(* IEC 61131-3 sources: TIA2AX/tests/V19/test_projects/expected/HW_2200330/ST20_PLC, 7 files *)

(* ---- HwIdentifiers.st ---- *)
TYPE
	HwIdentifiers : WORD
	(
		ST20_PLC_Profilschiene_0 :=	WORD#256,
		ST20_PLC :=	WORD#48,
		ST20_PLC_Card_reader_writer_1 :=	WORD#51,
		ST20_PLC_CPU_display_1 :=	WORD#54,
		ST20_PLC_OPC_UA_1 :=	WORD#117,
		ST20_PLC_DP_interface_1 :=	WORD#60,
		ST20_PLC_PROFINET_interface_1 :=	WORD#64,
		ST20_PLC_PROFINET_interface_1_Port_1 :=	WORD#65,
		ST20_PLC_PROFINET_interface_1_Port_2 :=	WORD#66,
		ST20_PLC_PROFINET_interface_2 :=	WORD#72,
		ST20_PLC_PROFINET_interface_2_Port_1 :=	WORD#73,
		ST20_Switch_SCALANCE_X_rack :=	WORD#544,
		ST20_Switch :=	WORD#545,
		ST20_Switch_ST20_Switch :=	WORD#546,
		ST20_Switch_SCALANCE_interface_1 :=	WORD#547,
		ST20_Switch_SCALANCE_interface_1_Port_1 :=	WORD#548,
		ST20_Switch_SCALANCE_interface_1_Port_2 :=	WORD#549,
		ST20_Switch_SCALANCE_interface_1_Port_3 :=	WORD#550,
		ST20_Switch_SCALANCE_interface_1_Port_4 :=	WORD#551,
		ST20_Switch_SCALANCE_interface_1_Port_5 :=	WORD#552,
		ST20_Switch_SCALANCE_interface_1_Port_6 :=	WORD#553,
		ST20_Switch_SCALANCE_interface_1_Port_7 :=	WORD#554,
		ST20_Switch_SCALANCE_interface_1_Port_8 :=	WORD#555,
		ST20_Switch_SCALANCE_interface_1_Port_9 :=	WORD#556,
		ST20_Switch_SCALANCE_interface_1_Port_10 :=	WORD#557,
		ST20_Switch_SCALANCE_interface_1_Port_11 :=	WORD#558,
		ST20_Switch_SCALANCE_interface_1_Port_12 :=	WORD#559,
		ST20_Switch_SCALANCE_interface_1_Port_13 :=	WORD#560,
		ST20_Switch_SCALANCE_interface_1_Port_14 :=	WORD#561,
		ST20_Switch_SCALANCE_interface_1_Port_15 :=	WORD#562,
		ST20_Switch_SCALANCE_interface_1_Port_16 :=	WORD#563,
		ST20_Switch_2_SCALANCE_X_rack :=	WORD#565,
		ST20_Switch_2 :=	WORD#566,
		ST20_Switch_2_ST20_Switch_2 :=	WORD#567,
		ST20_Switch_2_SCALANCE_interface_1 :=	WORD#568,
		ST20_Switch_2_SCALANCE_interface_1_Port_1 :=	WORD#569,
		ST20_Switch_2_SCALANCE_interface_1_Port_2 :=	WORD#570,
		ST20_Switch_2_SCALANCE_interface_1_Port_3 :=	WORD#571,
		ST20_Switch_2_SCALANCE_interface_1_Port_4 :=	WORD#572,
		ST20_Switch_2_SCALANCE_interface_1_Port_5 :=	WORD#573,
		ST20_Switch_2_SCALANCE_interface_1_Port_6 :=	WORD#574,
		ST20_Switch_2_SCALANCE_interface_1_Port_7 :=	WORD#575,
		ST20_Switch_2_SCALANCE_interface_1_Port_8 :=	WORD#576,
		ST20_Switch_2_SCALANCE_interface_1_Port_9 :=	WORD#577,
		ST20_Switch_2_SCALANCE_interface_1_Port_10 :=	WORD#578,
		ST20_Switch_2_SCALANCE_interface_1_Port_11 :=	WORD#579,
		ST20_Switch_2_SCALANCE_interface_1_Port_12 :=	WORD#580,
		ST20_Switch_2_SCALANCE_interface_1_Port_13 :=	WORD#581,
		ST20_Switch_2_SCALANCE_interface_1_Port_14 :=	WORD#582,
		ST20_Switch_2_SCALANCE_interface_1_Port_15 :=	WORD#583,
		ST20_Switch_2_SCALANCE_interface_1_Port_16 :=	WORD#584,
		ST20_Switch_3_SCALANCE_X_rack :=	WORD#586,
		ST20_Switch_3 :=	WORD#587,
		ST20_Switch_3_ST20_Switch_3 :=	WORD#588,
		ST20_Switch_3_SCALANCE_interface_1 :=	WORD#589,
		ST20_Switch_3_SCALANCE_interface_1_Port_1 :=	WORD#590,
		ST20_Switch_3_SCALANCE_interface_1_Port_2 :=	WORD#591,
		ST20_Switch_3_SCALANCE_interface_1_Port_3 :=	WORD#592,
		ST20_Switch_3_SCALANCE_interface_1_Port_4 :=	WORD#593,
		ST20_Switch_3_SCALANCE_interface_1_Port_5 :=	WORD#594,
		ST20_Switch_3_SCALANCE_interface_1_Port_6 :=	WORD#595,
		ST20_Switch_3_SCALANCE_interface_1_Port_7 :=	WORD#596,
		ST20_Switch_3_SCALANCE_interface_1_Port_8 :=	WORD#597,
		ST20_HMI_ConnectionBox_Connection_Box :=	WORD#265,
		ST20_HMI_ConnectionBox :=	WORD#258,
		ST20_HMI_ConnectionBox_ST20_HMI_ConnectionBox :=	WORD#259,
		ST20_HMI_ConnectionBox_SCALANCE_interface_1 :=	WORD#260,
		ST20_HMI_ConnectionBox_SCALANCE_interface_1_Port_1 :=	WORD#261,
		ST20_HMI_ConnectionBox_SCALANCE_interface_1_Port_2 :=	WORD#262,
		ST20_HMI_ConnectionBox_SCALANCE_interface_1_Port_3 :=	WORD#263,
		ST20_CPX_PN_IO_Interface :=	WORD#271,
		ST20_CPX_PN_IO_Interface_Port_1 :=	WORD#272,
		ST20_CPX_PN_IO_Interface_Port_2 :=	WORD#273,
		ST20_CPX_CPX :=	WORD#274,
		ST20_CPX_MPA1S_VMPA1_FB_EMS_8_8DO_1 :=	WORD#275,
		ST20_CPX_MPA1S_VMPA1_FB_EMS_8_8DO_2 :=	WORD#276,
		ST20_CPX_MPA1S_VMPA1_FB_EMS_8_8DO_3 :=	WORD#277,
		ST20_CPX_MPA1S_VMPA1_FB_EMS_8_8DO_4 :=	WORD#266,
		ST20_CPX_MPA1G_VMPA1_FB_EMG_8_8DO_1 :=	WORD#267,
		ST20_6_Promess_Rack :=	WORD#328,
		ST20_6_Promess :=	WORD#329,
		ST20_6_Promess_X1 :=	WORD#330,
		ST20_6_Promess_X1_X1_P1 :=	WORD#331,
		ST20_6_Promess_X1_X1_P2 :=	WORD#332,
		ST20_6_Promess_UniDrive_M :=	WORD#333,
		ST20_6_Promess_Menu_30_01_In_1 :=	WORD#334,
		ST20_6_Promess_Menu_30_02_In_1 :=	WORD#335,
		ST20_6_Promess_Menu_30_03_In_1 :=	WORD#336,
		ST20_6_Promess_Menu_30_04_In_1 :=	WORD#337,
		ST20_6_Promess_Menu_30_05_In_1 :=	WORD#338,
		ST20_6_Promess_Menu_30_06_In_1 :=	WORD#339,
		ST20_6_Promess_Menu_30_07_In_1 :=	WORD#340,
		ST20_6_Promess_Menu_30_08_In_1 :=	WORD#341,
		ST20_6_Promess_Menu_30_09_In_1 :=	WORD#342,
		ST20_6_Promess_Menu_30_10_In_1 :=	WORD#343,
		ST20_6_Promess_Menu_30_11_In_1 :=	WORD#344,
		ST20_6_Promess_Menu_30_12_In_1 :=	WORD#345,
		ST20_6_Promess_Menu_30_13_In_1 :=	WORD#346,
		ST20_6_Promess_Menu_30_14_In_1 :=	WORD#347,
		ST20_6_Promess_Menu_30_15_In_1 :=	WORD#348,
		ST20_6_Promess_Menu_30_16_In_1 :=	WORD#278,
		ST20_6_Promess_Menu_30_33_Out_1 :=	WORD#279,
		ST20_6_Promess_Menu_30_34_Out_1 :=	WORD#280,
		ST20_6_Promess_Menu_30_35_Out_1 :=	WORD#281,
		ST20_6_Promess_Menu_30_36_Out_1 :=	WORD#282,
		ST20_6_Promess_Menu_30_37_Out_1 :=	WORD#283,
		ST20_6_Promess_Menu_30_38_Out_1 :=	WORD#284,
		ST20_6_Promess_Menu_30_39_Out_1 :=	WORD#285,
		ST20_6_Promess_Menu_30_40_Out_1 :=	WORD#286,
		ST20_6_Promess_Menu_30_41_Out_1 :=	WORD#287,
		ST20_6_Promess_Menu_30_42_Out_1 :=	WORD#288,
		ST20_6_Promess_Menu_30_43_Out_1 :=	WORD#289,
		ST20_6_Promess_Menu_30_44_Out_1 :=	WORD#290,
		ST20_6_Promess_Menu_30_45_Out_1 :=	WORD#291,
		ST20_6_Promess_Menu_30_46_Out_1 :=	WORD#292,
		ST20_6_Promess_Menu_30_47_Out_1 :=	WORD#293,
		ST20_6_Promess_Menu_30_48_Out_1 :=	WORD#294,
		ST20_6_Promess_Menu_30_17_In_1 :=	WORD#295,
		ST20_6_Promess_Menu_30_18_In_1 :=	WORD#296,
		ST20_6_Promess_Menu_30_19_In_1 :=	WORD#297,
		ST20_6_Promess_Menu_30_20_In_1 :=	WORD#298,
		ST20_6_Promess_Menu_30_21_In_1 :=	WORD#299,
		ST20_6_Promess_Menu_30_22_In_1 :=	WORD#300,
		ST20_6_Promess_Menu_30_23_In_1 :=	WORD#301,
		ST20_6_Promess_Menu_30_24_In_1 :=	WORD#302,
		ST20_6_Promess_Menu_30_25_In_1 :=	WORD#303,
		ST20_6_Promess_Menu_30_26_In_1 :=	WORD#304,
		ST20_6_Promess_Menu_30_27_In_1 :=	WORD#305,
		ST20_6_Promess_Menu_30_28_In_1 :=	WORD#306,
		ST20_6_Promess_Menu_30_29_In_1 :=	WORD#307,
		ST20_6_Promess_Menu_30_30_In_1 :=	WORD#308,
		ST20_6_Promess_Menu_30_31_In_1 :=	WORD#309,
		ST20_6_Promess_Menu_30_32_In_1 :=	WORD#310,
		ST20_6_Promess_Menu_30_49_Out_1 :=	WORD#311,
		ST20_6_Promess_Menu_30_50_Out_1 :=	WORD#312,
		ST20_6_Promess_Menu_30_51_Out_1 :=	WORD#313,
		ST20_6_Promess_Menu_30_52_Out_1 :=	WORD#314,
		ST20_6_Promess_Menu_30_53_Out_1 :=	WORD#315,
		ST20_6_Promess_Menu_30_54_Out_1 :=	WORD#316,
		ST20_6_Promess_Menu_30_55_Out_1 :=	WORD#317,
		ST20_6_Promess_Menu_30_56_Out_1 :=	WORD#318,
		ST20_6_Promess_Menu_30_57_Out_1 :=	WORD#319,
		ST20_6_Promess_Menu_30_58_Out_1 :=	WORD#320,
		ST20_6_Promess_Menu_30_59_Out_1 :=	WORD#321,
		ST20_6_Promess_Menu_30_60_Out_1 :=	WORD#322,
		ST20_6_Promess_Menu_30_61_Out_1 :=	WORD#323,
		ST20_6_Promess_Menu_30_62_Out_1 :=	WORD#324,
		ST20_6_Promess_Menu_30_63_Out_1 :=	WORD#325,
		ST20_6_Promess_Menu_30_64_Out_1 :=	WORD#326,
		ST20_7_CMMT_3GF1_PN_IO_Interface :=	WORD#352,
		ST20_7_CMMT_3GF1_PN_IO_Interface_Port_1 :=	WORD#353,
		ST20_7_CMMT_3GF1_PN_IO_Interface_Port_2 :=	WORD#354,
		ST20_7_CMMT_3GF1_CMMT_AS_V1 :=	WORD#355,
		ST20_7_CMMT_3GF1_DO_SERVO_1_Module_Access_Point :=	WORD#357,
		ST20_7_CMMT_3GF1_DO_SERVO_1_Siemens_telegram_111_PZD_12_12 :=	WORD#358,
		ST20_7_CMMT_3GF1_Siemens_telegram_111_PZD_12_12 :=	WORD#358,
		ST20_1_DM260_Rack :=	WORD#360,
		ST20_1_DM260 :=	WORD#361,
		ST20_1_DM260_Interface :=	WORD#362,
		ST20_1_DM260_Interface_Port_1 :=	WORD#363,
		ST20_1_DM260_DataMan_260 :=	WORD#364,
		ST20_1_DM260_Acquisition_Control_1 :=	WORD#365,
		ST20_1_DM260_Acquisition_Status_1 :=	WORD#366,
		ST20_1_DM260_Results_Control_1 :=	WORD#367,
		ST20_1_DM260_Results_Status_1 :=	WORD#368,
		ST20_1_DM260_Soft_Event_Control_1 :=	WORD#369,
		ST20_1_DM260_User_Data_64_bytes_1 :=	WORD#370,
		ST20_1_DM260_Result_Data_64_bytes_1 :=	WORD#371,
		ST20_5_DM260_Rack :=	WORD#373,
		ST20_5_DM260 :=	WORD#374,
		ST20_5_DM260_Interface :=	WORD#375,
		ST20_5_DM260_Interface_Port_1 :=	WORD#376,
		ST20_5_DM260_DataMan_260 :=	WORD#377,
		ST20_5_DM260_Acquisition_Control_1 :=	WORD#378,
		ST20_5_DM260_Acquisition_Status_1 :=	WORD#379,
		ST20_5_DM260_Results_Control_1 :=	WORD#380,
		ST20_5_DM260_Results_Status_1 :=	WORD#381,
		ST20_5_DM260_Soft_Event_Control_1 :=	WORD#382,
		ST20_5_DM260_User_Data_64_bytes_1 :=	WORD#383,
		ST20_5_DM260_Result_Data_64_bytes_1 :=	WORD#384,
		ST20_2_DM260_Rack :=	WORD#386,
		ST20_2_DM260 :=	WORD#387,
		ST20_2_DM260_Interface :=	WORD#388,
		ST20_2_DM260_Interface_Port_1 :=	WORD#389,
		ST20_2_DM260_DataMan_260 :=	WORD#390,
		ST20_2_DM260_Acquisition_Control_1 :=	WORD#391,
		ST20_2_DM260_Acquisition_Status_1 :=	WORD#392,
		ST20_2_DM260_Results_Control_1 :=	WORD#393,
		ST20_2_DM260_Results_Status_1 :=	WORD#394,
		ST20_2_DM260_Soft_Event_Control_1 :=	WORD#395,
		ST20_2_DM260_User_Data_64_bytes_1 :=	WORD#396,
		ST20_2_DM260_Result_Data_64_bytes_1 :=	WORD#397,
		ST20_2_TZ535_PN_Rack :=	WORD#399,
		ST20_2_TZ535_PN :=	WORD#400,
		ST20_2_TZ535_PN_Interface :=	WORD#401,
		ST20_2_TZ535_PN_Interface_Port_1 :=	WORD#402,
		ST20_2_TZ535_PN_Interface_Port_2 :=	WORD#403,
		ST20_2_TZ535_PN_2D_TZ535_PN_PROFINET_IO :=	WORD#404,
		ST20_2_TZ535_PN_In_Out_32_byte_1 :=	WORD#405,
		ST20_3_TZ535_PN_Rack :=	WORD#407,
		ST20_3_TZ535_PN :=	WORD#408,
		ST20_3_TZ535_PN_Interface :=	WORD#409,
		ST20_3_TZ535_PN_Interface_Port_1 :=	WORD#410,
		ST20_3_TZ535_PN_Interface_Port_2 :=	WORD#411,
		ST20_3_TZ535_PN_2D_TZ535_PN_PROFINET_IO :=	WORD#412,
		ST20_3_TZ535_PN_In_Out_32_byte_1 :=	WORD#413,
		ST20_4_TZ535_PN_Rack :=	WORD#415,
		ST20_4_TZ535_PN :=	WORD#416,
		ST20_4_TZ535_PN_Interface :=	WORD#417,
		ST20_4_TZ535_PN_Interface_Port_1 :=	WORD#418,
		ST20_4_TZ535_PN_Interface_Port_2 :=	WORD#419,
		ST20_4_TZ535_PN_2D_TZ535_PN_PROFINET_IO :=	WORD#420,
		ST20_4_TZ535_PN_In_Out_32_byte_1 :=	WORD#421,
		ST20_5_TZ535_PN_Rack :=	WORD#423,
		ST20_5_TZ535_PN :=	WORD#424,
		ST20_5_TZ535_PN_Interface :=	WORD#425,
		ST20_5_TZ535_PN_Interface_Port_1 :=	WORD#426,
		ST20_5_TZ535_PN_Interface_Port_2 :=	WORD#427,
		ST20_5_TZ535_PN_2D_TZ535_PN_PROFINET_IO :=	WORD#428,
		ST20_5_TZ535_PN_In_Out_32_byte_1 :=	WORD#429,
		ST20_ET200SP_Rack_0 :=	WORD#431,
		ST20_ET200SP :=	WORD#432,
		ST20_ET200SP_ST20_ET200SP :=	WORD#433,
		ST20_ET200SP_PROFINET_interface :=	WORD#434,
		ST20_ET200SP_PROFINET_interface_Port_1 :=	WORD#436,
		ST20_ET200SP_PROFINET_interface_Port_2 :=	WORD#435,
		ST20_ET200SP_BA_2xRJ45 :=	WORD#436,
		ST20_ET200SP_CM_4xIO_Link_1 :=	WORD#437,
		ST20_ET200SP_CM_4xIO_Link_2 :=	WORD#438,
		ST20_ET200SP_DI_16x24VDC_ST_1 :=	WORD#439,
		ST20_ET200SP_DI_16x24VDC_ST_2 :=	WORD#440,
		ST20_ET200SP_DI_16x24VDC_ST_3 :=	WORD#441,
		ST20_ET200SP_DI_16x24VDC_ST_4 :=	WORD#442,
		ST20_ET200SP_DQ_16x24VDC_0_5A_ST_1 :=	WORD#443,
		ST20_ET200SP_DQ_16x24VDC_0_5A_ST_2 :=	WORD#444,
		ST20_ET200SP_DQ_16x24VDC_0_5A_ST_3 :=	WORD#445,
		ST20_ET200SP_Servermodul_1 :=	WORD#446,
		ST20_2_Schunk_Rack :=	WORD#448,
		ST20_2_Schunk :=	WORD#449,
		ST20_2_Schunk_Interface :=	WORD#450,
		ST20_2_Schunk_Interface_Port_1 :=	WORD#451,
		ST20_2_Schunk_Interface_Port_2 :=	WORD#452,
		ST20_2_Schunk_DEVICE_SFP :=	WORD#453,
		ST20_2_Schunk_IN_4_Double_Words_1 :=	WORD#454,
		ST20_2_Schunk_OUT_4_Double_Words_1 :=	WORD#455,
		ST20_5_Schunk_Rack :=	WORD#457,
		ST20_5_Schunk :=	WORD#458,
		ST20_5_Schunk_Interface :=	WORD#459,
		ST20_5_Schunk_Interface_Port_1 :=	WORD#460,
		ST20_5_Schunk_Interface_Port_2 :=	WORD#461,
		ST20_5_Schunk_DEVICE_SFP :=	WORD#462,
		ST20_5_Schunk_IN_4_Double_Words_1 :=	WORD#463,
		ST20_5_Schunk_OUT_4_Double_Words_1 :=	WORD#464,
		ST20_2_DM260_PCB1_Rack :=	WORD#466,
		ST20_2_DM260_PCB1 :=	WORD#467,
		ST20_2_DM260_PCB1_Interface :=	WORD#468,
		ST20_2_DM260_PCB1_Interface_Port_1 :=	WORD#469,
		ST20_2_DM260_PCB1_DataMan_260 :=	WORD#470,
		ST20_2_DM260_PCB1_Acquisition_Control_1 :=	WORD#471,
		ST20_2_DM260_PCB1_Acquisition_Status_1 :=	WORD#472,
		ST20_2_DM260_PCB1_Results_Control_1 :=	WORD#473,
		ST20_2_DM260_PCB1_Results_Status_1 :=	WORD#474,
		ST20_2_DM260_PCB1_Soft_Event_Control_1 :=	WORD#475,
		ST20_2_DM260_PCB1_User_Data_64_bytes_1 :=	WORD#476,
		ST20_2_DM260_PCB1_Result_Data_64_bytes_1 :=	WORD#477,
		ST20_2_DM260_PCB2_Rack :=	WORD#479,
		ST20_2_DM260_PCB2 :=	WORD#480,
		ST20_2_DM260_PCB2_Interface :=	WORD#481,
		ST20_2_DM260_PCB2_Interface_Port_1 :=	WORD#482,
		ST20_2_DM260_PCB2_DataMan_260 :=	WORD#483,
		ST20_2_DM260_PCB2_Acquisition_Control_1 :=	WORD#484,
		ST20_2_DM260_PCB2_Acquisition_Status_1 :=	WORD#485,
		ST20_2_DM260_PCB2_Results_Control_1 :=	WORD#486,
		ST20_2_DM260_PCB2_Results_Status_1 :=	WORD#487,
		ST20_2_DM260_PCB2_Soft_Event_Control_1 :=	WORD#488,
		ST20_2_DM260_PCB2_User_Data_64_bytes_1 :=	WORD#489,
		ST20_2_DM260_PCB2_Result_Data_64_bytes_1 :=	WORD#490,
		ST20_CPX_2_PN_IO_Interface :=	WORD#494,
		ST20_CPX_2_PN_IO_Interface_Port_1 :=	WORD#495,
		ST20_CPX_2_PN_IO_Interface_Port_2 :=	WORD#496,
		ST20_CPX_2_CPX :=	WORD#497,
		ST20_CPX_2_MPA1S_VMPA1_FB_EMS_8_8DO_1 :=	WORD#498,
		ST20_CPX_2_MPA1S_VMPA1_FB_EMS_8_8DO_2 :=	WORD#499,
		ST20_CPX_2_MPA1G_VMPA1_FB_EMG_8_8DO_1 :=	WORD#500,
		ST20_CPX_2_MPA1G_VMPA1_FB_EMG_8_8DO_2 :=	WORD#501,
		ST20_3_Schunk_Rack :=	WORD#503,
		ST20_3_Schunk :=	WORD#504,
		ST20_3_Schunk_Interface :=	WORD#505,
		ST20_3_Schunk_Interface_Port_1 :=	WORD#506,
		ST20_3_Schunk_Interface_Port_2 :=	WORD#507,
		ST20_3_Schunk_DEVICE_SFP :=	WORD#508,
		ST20_3_Schunk_IN_4_Double_Words_1 :=	WORD#509,
		ST20_3_Schunk_OUT_4_Double_Words_1 :=	WORD#510,
		ST20_4_Schunk_Rack :=	WORD#512,
		ST20_4_Schunk :=	WORD#513,
		ST20_4_Schunk_Interface :=	WORD#514,
		ST20_4_Schunk_Interface_Port_1 :=	WORD#515,
		ST20_4_Schunk_Interface_Port_2 :=	WORD#516,
		ST20_4_Schunk_DEVICE_SFP :=	WORD#517,
		ST20_4_Schunk_IN_4_Double_Words_1 :=	WORD#518,
		ST20_4_Schunk_OUT_4_Double_Words_1 :=	WORD#519,
		ST20_1_md_u2xxx_Rack :=	WORD#521,
		ST20_1_md_u2xxx :=	WORD#522,
		ST20_1_md_u2xxx_Interface :=	WORD#523,
		ST20_1_md_u2xxx_Interface_Port_1 :=	WORD#524,
		ST20_1_md_u2xxx_MD_X2XXX :=	WORD#525,
		ST20_1_md_u2xxx_Machine_Status_1 :=	WORD#526,
		ST20_1_md_u2xxx_Function_Status_1 :=	WORD#527,
		ST20_1_md_u2xxx_Completion_Status_1 :=	WORD#528,
		ST20_1_md_u2xxx_Error_Status_1 :=	WORD#529,
		ST20_1_md_u2xxx_Error_Codes_1 :=	WORD#530,
		ST20_1_md_u2xxx_Operate_Parametere_1 :=	WORD#531,
		ST20_1_md_u2xxx_2D_Code_Read_Result_1 :=	WORD#532,
		ST20_1_md_u2xxx_Count_Result_Data_1 :=	WORD#533,
		ST20_1_md_u2xxx_Result_Data_128byte_1 :=	WORD#534,
		ST20_1_md_u2xxx_General_Request_1 :=	WORD#535,
		ST20_1_md_u2xxx_Function_Request_1 :=	WORD#536,
		ST20_1_md_u2xxx_Request_Completion_Clear_1 :=	WORD#537,
		ST20_1_md_u2xxx_Request_Parameter_1 :=	WORD#538,
		ST20_1_md_u2xxx_Request_Data_128byte_1 :=	WORD#539,
		NONE:= WORD#0
	);
END_TYPE

(* ---- HwInputs.st ---- *)
TYPE
	HwInputs : STRUCT
		ST20_6_Promess_Menu_30_01_In_1 AT %B2100 : WORD;
		ST20_6_Promess_Menu_30_02_In_1 AT %B2102 : WORD;
		ST20_6_Promess_Menu_30_03_In_1 AT %B2104 : WORD;
		ST20_6_Promess_Menu_30_04_In_1 AT %B2106 : WORD;
		ST20_6_Promess_Menu_30_05_In_1 AT %B2108 : WORD;
		ST20_6_Promess_Menu_30_06_In_1 AT %B2110 : WORD;
		ST20_6_Promess_Menu_30_07_In_1 AT %B2112 : WORD;
		ST20_6_Promess_Menu_30_08_In_1 AT %B2114 : WORD;
		ST20_6_Promess_Menu_30_09_In_1 AT %B2116 : WORD;
		ST20_6_Promess_Menu_30_10_In_1 AT %B2118 : WORD;
		ST20_6_Promess_Menu_30_11_In_1 AT %B2120 : WORD;
		ST20_6_Promess_Menu_30_12_In_1 AT %B2122 : WORD;
		ST20_6_Promess_Menu_30_13_In_1 AT %B2124 : WORD;
		ST20_6_Promess_Menu_30_14_In_1 AT %B2126 : WORD;
		ST20_6_Promess_Menu_30_15_In_1 AT %B2128 : WORD;
		ST20_6_Promess_Menu_30_16_In_1 AT %B2130 : WORD;
		ST20_6_Promess_Menu_30_17_In_1 AT %B2132 : WORD;
		ST20_6_Promess_Menu_30_18_In_1 AT %B2134 : WORD;
		ST20_6_Promess_Menu_30_19_In_1 AT %B2136 : WORD;
		ST20_6_Promess_Menu_30_20_In_1 AT %B2138 : WORD;
		ST20_6_Promess_Menu_30_21_In_1 AT %B2140 : WORD;
		ST20_6_Promess_Menu_30_22_In_1 AT %B2142 : WORD;
		ST20_6_Promess_Menu_30_23_In_1 AT %B2144 : WORD;
		ST20_6_Promess_Menu_30_24_In_1 AT %B2146 : WORD;
		ST20_6_Promess_Menu_30_25_In_1 AT %B2148 : WORD;
		ST20_6_Promess_Menu_30_26_In_1 AT %B2150 : WORD;
		ST20_6_Promess_Menu_30_27_In_1 AT %B2152 : WORD;
		ST20_6_Promess_Menu_30_28_In_1 AT %B2154 : WORD;
		ST20_6_Promess_Menu_30_29_In_1 AT %B2156 : WORD;
		ST20_6_Promess_Menu_30_30_In_1 AT %B2158 : WORD;
		ST20_6_Promess_Menu_30_31_In_1 AT %B2160 : WORD;
		ST20_6_Promess_Menu_30_32_In_1 AT %B2162 : WORD;
		ST20_7_CMMT_3GF1_DO_SERVO_1_Siemens_telegram_111_PZD_12_12 AT %B7100 : ARRAY[0..23] OF BYTE;
		ST20_1_DM260_Acquisition_Status_1 AT %B1000 : ARRAY[0..2] OF BYTE;
		ST20_1_DM260_Results_Status_1 AT %B1003 : BYTE;
		ST20_1_DM260_Soft_Event_Control_1 AT %B1004 : BYTE;
		ST20_1_DM260_Result_Data_64_bytes_1 AT %B1010 : ARRAY[0..71] OF BYTE;
		ST20_5_DM260_Acquisition_Status_1 AT %B5000 : ARRAY[0..2] OF BYTE;
		ST20_5_DM260_Results_Status_1 AT %B5003 : BYTE;
		ST20_5_DM260_Soft_Event_Control_1 AT %B5004 : BYTE;
		ST20_5_DM260_Result_Data_64_bytes_1 AT %B5010 : ARRAY[0..71] OF BYTE;
		ST20_2_DM260_Acquisition_Status_1 AT %B2000 : ARRAY[0..2] OF BYTE;
		ST20_2_DM260_Results_Status_1 AT %B2003 : BYTE;
		ST20_2_DM260_Soft_Event_Control_1 AT %B2004 : BYTE;
		ST20_2_DM260_Result_Data_64_bytes_1 AT %B2010 : ARRAY[0..71] OF BYTE;
		ST20_2_TZ535_PN_In_Out_32_byte_1 AT %B2500 : ARRAY[0..31] OF BYTE;
		ST20_3_TZ535_PN_In_Out_32_byte_1 AT %B3500 : ARRAY[0..31] OF BYTE;
		ST20_4_TZ535_PN_In_Out_32_byte_1 AT %B4500 : ARRAY[0..31] OF BYTE;
		ST20_5_TZ535_PN_In_Out_32_byte_1 AT %B5500 : ARRAY[0..31] OF BYTE;
		ST20_ET200SP_CM_4xIO_Link_1 AT %B100 : ARRAY[0..31] OF BYTE;
		ST20_ET200SP_CM_4xIO_Link_2 AT %B132 : ARRAY[0..31] OF BYTE;
		ST20_ET200SP_DI_16x24VDC_ST_1 AT %B0 : WORD;
		ST20_ET200SP_DI_16x24VDC_ST_2 AT %B2 : WORD;
		ST20_ET200SP_DI_16x24VDC_ST_3 AT %B4 : WORD;
		ST20_ET200SP_DI_16x24VDC_ST_4 AT %B6 : WORD;
		ST20_2_Schunk_IN_4_Double_Words_1 AT %B2600 : ARRAY[0..15] OF BYTE;
		ST20_5_Schunk_IN_4_Double_Words_1 AT %B5600 : ARRAY[0..15] OF BYTE;
		ST20_2_DM260_PCB1_Acquisition_Status_1 AT %B2300 : ARRAY[0..2] OF BYTE;
		ST20_2_DM260_PCB1_Results_Status_1 AT %B2303 : BYTE;
		ST20_2_DM260_PCB1_Soft_Event_Control_1 AT %B2304 : BYTE;
		ST20_2_DM260_PCB1_Result_Data_64_bytes_1 AT %B2310 : ARRAY[0..71] OF BYTE;
		ST20_2_DM260_PCB2_Acquisition_Status_1 AT %B2005 : ARRAY[0..2] OF BYTE;
		ST20_2_DM260_PCB2_Results_Status_1 AT %B2008 : BYTE;
		ST20_2_DM260_PCB2_Soft_Event_Control_1 AT %B2009 : BYTE;
		ST20_2_DM260_PCB2_Result_Data_64_bytes_1 AT %B2164 : ARRAY[0..71] OF BYTE;
		ST20_3_Schunk_IN_4_Double_Words_1 AT %B2616 : ARRAY[0..15] OF BYTE;
		ST20_4_Schunk_IN_4_Double_Words_1 AT %B2632 : ARRAY[0..15] OF BYTE;
		ST20_1_md_u2xxx_Machine_Status_1 AT %B20 : DWORD;
		ST20_1_md_u2xxx_Function_Status_1 AT %B24 : DWORD;
		ST20_1_md_u2xxx_Completion_Status_1 AT %B74 : ARRAY[0..7] OF BYTE;
		ST20_1_md_u2xxx_Error_Status_1 AT %B196 : ARRAY[0..7] OF BYTE;
		ST20_1_md_u2xxx_Error_Codes_1 AT %B204 : ARRAY[0..7] OF BYTE;
		ST20_1_md_u2xxx_Operate_Parametere_1 AT %B212 : ARRAY[0..15] OF BYTE;
		ST20_1_md_u2xxx_2D_Code_Read_Result_1 AT %B292 : ARRAY[0..7] OF BYTE;
		ST20_1_md_u2xxx_Count_Result_Data_1 AT %B300 : DWORD;
		ST20_1_md_u2xxx_Result_Data_128byte_1 AT %B304 : ARRAY[0..129] OF BYTE;
	END_STRUCT;
END_TYPE

(* ---- HwOutputs.st ---- *)
TYPE
	HwOutputs : STRUCT
		ST20_CPX_MPA1S_VMPA1_FB_EMS_8_8DO_1 AT %B200 : BYTE;
		ST20_CPX_MPA1S_VMPA1_FB_EMS_8_8DO_2 AT %B201 : BYTE;
		ST20_CPX_MPA1S_VMPA1_FB_EMS_8_8DO_3 AT %B202 : BYTE;
		ST20_CPX_MPA1S_VMPA1_FB_EMS_8_8DO_4 AT %B203 : BYTE;
		ST20_CPX_MPA1G_VMPA1_FB_EMG_8_8DO_1 AT %B204 : BYTE;
		ST20_6_Promess_Menu_30_33_Out_1 AT %B2100 : WORD;
		ST20_6_Promess_Menu_30_34_Out_1 AT %B2102 : WORD;
		ST20_6_Promess_Menu_30_35_Out_1 AT %B2104 : WORD;
		ST20_6_Promess_Menu_30_36_Out_1 AT %B2106 : WORD;
		ST20_6_Promess_Menu_30_37_Out_1 AT %B2108 : WORD;
		ST20_6_Promess_Menu_30_38_Out_1 AT %B2110 : WORD;
		ST20_6_Promess_Menu_30_39_Out_1 AT %B2112 : WORD;
		ST20_6_Promess_Menu_30_40_Out_1 AT %B2114 : WORD;
		ST20_6_Promess_Menu_30_41_Out_1 AT %B2116 : WORD;
		ST20_6_Promess_Menu_30_42_Out_1 AT %B2118 : WORD;
		ST20_6_Promess_Menu_30_43_Out_1 AT %B2120 : WORD;
		ST20_6_Promess_Menu_30_44_Out_1 AT %B2122 : WORD;
		ST20_6_Promess_Menu_30_45_Out_1 AT %B2124 : WORD;
		ST20_6_Promess_Menu_30_46_Out_1 AT %B2126 : WORD;
		ST20_6_Promess_Menu_30_47_Out_1 AT %B2128 : WORD;
		ST20_6_Promess_Menu_30_48_Out_1 AT %B2130 : WORD;
		ST20_6_Promess_Menu_30_49_Out_1 AT %B2132 : WORD;
		ST20_6_Promess_Menu_30_50_Out_1 AT %B2134 : WORD;
		ST20_6_Promess_Menu_30_51_Out_1 AT %B2136 : WORD;
		ST20_6_Promess_Menu_30_52_Out_1 AT %B2138 : WORD;
		ST20_6_Promess_Menu_30_53_Out_1 AT %B2140 : WORD;
		ST20_6_Promess_Menu_30_54_Out_1 AT %B2142 : WORD;
		ST20_6_Promess_Menu_30_55_Out_1 AT %B2144 : WORD;
		ST20_6_Promess_Menu_30_56_Out_1 AT %B2146 : WORD;
		ST20_6_Promess_Menu_30_57_Out_1 AT %B2148 : WORD;
		ST20_6_Promess_Menu_30_58_Out_1 AT %B2150 : WORD;
		ST20_6_Promess_Menu_30_59_Out_1 AT %B2152 : WORD;
		ST20_6_Promess_Menu_30_60_Out_1 AT %B2154 : WORD;
		ST20_6_Promess_Menu_30_61_Out_1 AT %B2156 : WORD;
		ST20_6_Promess_Menu_30_62_Out_1 AT %B2158 : WORD;
		ST20_6_Promess_Menu_30_63_Out_1 AT %B2160 : WORD;
		ST20_6_Promess_Menu_30_64_Out_1 AT %B2162 : WORD;
		ST20_7_CMMT_3GF1_DO_SERVO_1_Siemens_telegram_111_PZD_12_12 AT %B7100 : ARRAY[0..23] OF BYTE;
		ST20_1_DM260_Acquisition_Control_1 AT %B1000 : BYTE;
		ST20_1_DM260_Results_Control_1 AT %B1003 : BYTE;
		ST20_1_DM260_Soft_Event_Control_1 AT %B1004 : BYTE;
		ST20_1_DM260_User_Data_64_bytes_1 AT %B1010 : ARRAY[0..67] OF BYTE;
		ST20_5_DM260_Acquisition_Control_1 AT %B5000 : BYTE;
		ST20_5_DM260_Results_Control_1 AT %B5003 : BYTE;
		ST20_5_DM260_Soft_Event_Control_1 AT %B5004 : BYTE;
		ST20_5_DM260_User_Data_64_bytes_1 AT %B5010 : ARRAY[0..67] OF BYTE;
		ST20_2_DM260_Acquisition_Control_1 AT %B2000 : BYTE;
		ST20_2_DM260_Results_Control_1 AT %B2003 : BYTE;
		ST20_2_DM260_Soft_Event_Control_1 AT %B2004 : BYTE;
		ST20_2_DM260_User_Data_64_bytes_1 AT %B2010 : ARRAY[0..67] OF BYTE;
		ST20_2_TZ535_PN_In_Out_32_byte_1 AT %B2500 : ARRAY[0..31] OF BYTE;
		ST20_3_TZ535_PN_In_Out_32_byte_1 AT %B3500 : ARRAY[0..31] OF BYTE;
		ST20_4_TZ535_PN_In_Out_32_byte_1 AT %B4500 : ARRAY[0..31] OF BYTE;
		ST20_5_TZ535_PN_In_Out_32_byte_1 AT %B5500 : ARRAY[0..31] OF BYTE;
		ST20_ET200SP_CM_4xIO_Link_1 AT %B100 : ARRAY[0..31] OF BYTE;
		ST20_ET200SP_CM_4xIO_Link_2 AT %B132 : ARRAY[0..31] OF BYTE;
		ST20_ET200SP_DQ_16x24VDC_0_5A_ST_1 AT %B0 : WORD;
		ST20_ET200SP_DQ_16x24VDC_0_5A_ST_2 AT %B2 : WORD;
		ST20_ET200SP_DQ_16x24VDC_0_5A_ST_3 AT %B4 : WORD;
		ST20_2_Schunk_OUT_4_Double_Words_1 AT %B2600 : ARRAY[0..15] OF BYTE;
		ST20_5_Schunk_OUT_4_Double_Words_1 AT %B5600 : ARRAY[0..15] OF BYTE;
		ST20_2_DM260_PCB1_Acquisition_Control_1 AT %B2300 : BYTE;
		ST20_2_DM260_PCB1_Results_Control_1 AT %B2303 : BYTE;
		ST20_2_DM260_PCB1_Soft_Event_Control_1 AT %B2304 : BYTE;
		ST20_2_DM260_PCB1_User_Data_64_bytes_1 AT %B2310 : ARRAY[0..67] OF BYTE;
		ST20_2_DM260_PCB2_Acquisition_Control_1 AT %B2001 : BYTE;
		ST20_2_DM260_PCB2_Results_Control_1 AT %B2005 : BYTE;
		ST20_2_DM260_PCB2_Soft_Event_Control_1 AT %B2006 : BYTE;
		ST20_2_DM260_PCB2_User_Data_64_bytes_1 AT %B2164 : ARRAY[0..67] OF BYTE;
		ST20_CPX_2_MPA1S_VMPA1_FB_EMS_8_8DO_1 AT %B210 : BYTE;
		ST20_CPX_2_MPA1S_VMPA1_FB_EMS_8_8DO_2 AT %B211 : BYTE;
		ST20_CPX_2_MPA1G_VMPA1_FB_EMG_8_8DO_1 AT %B212 : BYTE;
		ST20_CPX_2_MPA1G_VMPA1_FB_EMG_8_8DO_2 AT %B213 : BYTE;
		ST20_3_Schunk_OUT_4_Double_Words_1 AT %B2616 : ARRAY[0..15] OF BYTE;
		ST20_4_Schunk_OUT_4_Double_Words_1 AT %B2632 : ARRAY[0..15] OF BYTE;
		ST20_1_md_u2xxx_General_Request_1 AT %B16 : ARRAY[0..7] OF BYTE;
		ST20_1_md_u2xxx_Function_Request_1 AT %B24 : DWORD;
		ST20_1_md_u2xxx_Request_Completion_Clear_1 AT %B74 : ARRAY[0..7] OF BYTE;
		ST20_1_md_u2xxx_Request_Parameter_1 AT %B82 : DWORD;
		ST20_1_md_u2xxx_Request_Data_128byte_1 AT %B311 : ARRAY[0..129] OF BYTE;
	END_STRUCT;
END_TYPE

(* ---- PlcInputs.st ---- *)
TYPE
	PlcInputs : STRUCT
		ST20_6_Promess_Menu_30_01_In_1 : WORD;
		ST20_6_Promess_Menu_30_02_In_1 : WORD;
		ST20_6_Promess_Menu_30_03_In_1 : WORD;
		ST20_6_Promess_Menu_30_04_In_1 : WORD;
		ST20_6_Promess_Menu_30_05_In_1 : WORD;
		ST20_6_Promess_Menu_30_06_In_1 : WORD;
		ST20_6_Promess_Menu_30_07_In_1 : WORD;
		ST20_6_Promess_Menu_30_08_In_1 : WORD;
		ST20_6_Promess_Menu_30_09_In_1 : WORD;
		ST20_6_Promess_Menu_30_10_In_1 : WORD;
		ST20_6_Promess_Menu_30_11_In_1 : WORD;
		ST20_6_Promess_Menu_30_12_In_1 : WORD;
		ST20_6_Promess_Menu_30_13_In_1 : WORD;
		ST20_6_Promess_Menu_30_14_In_1 : WORD;
		ST20_6_Promess_Menu_30_15_In_1 : WORD;
		ST20_6_Promess_Menu_30_16_In_1 : WORD;
		ST20_6_Promess_Menu_30_17_In_1 : WORD;
		ST20_6_Promess_Menu_30_18_In_1 : WORD;
		ST20_6_Promess_Menu_30_19_In_1 : WORD;
		ST20_6_Promess_Menu_30_20_In_1 : WORD;
		ST20_6_Promess_Menu_30_21_In_1 : WORD;
		ST20_6_Promess_Menu_30_22_In_1 : WORD;
		ST20_6_Promess_Menu_30_23_In_1 : WORD;
		ST20_6_Promess_Menu_30_24_In_1 : WORD;
		ST20_6_Promess_Menu_30_25_In_1 : WORD;
		ST20_6_Promess_Menu_30_26_In_1 : WORD;
		ST20_6_Promess_Menu_30_27_In_1 : WORD;
		ST20_6_Promess_Menu_30_28_In_1 : WORD;
		ST20_6_Promess_Menu_30_29_In_1 : WORD;
		ST20_6_Promess_Menu_30_30_In_1 : WORD;
		ST20_6_Promess_Menu_30_31_In_1 : WORD;
		ST20_6_Promess_Menu_30_32_In_1 : WORD;
		ST20_7_CMMT_3GF1_DO_SERVO_1_Siemens_telegram_111_PZD_12_12 : ARRAY[0..23] OF BYTE;
		ST20_1_DM260_Acquisition_Status_1 : ARRAY[0..2] OF BYTE;
		ST20_1_DM260_Results_Status_1 : BYTE;
		ST20_1_DM260_Soft_Event_Control_1 : BYTE;
		ST20_1_DM260_Result_Data_64_bytes_1 : ARRAY[0..71] OF BYTE;
		ST20_5_DM260_Acquisition_Status_1 : ARRAY[0..2] OF BYTE;
		ST20_5_DM260_Results_Status_1 : BYTE;
		ST20_5_DM260_Soft_Event_Control_1 : BYTE;
		ST20_5_DM260_Result_Data_64_bytes_1 : ARRAY[0..71] OF BYTE;
		ST20_2_DM260_Acquisition_Status_1 : ARRAY[0..2] OF BYTE;
		ST20_2_DM260_Results_Status_1 : BYTE;
		ST20_2_DM260_Soft_Event_Control_1 : BYTE;
		ST20_2_DM260_Result_Data_64_bytes_1 : ARRAY[0..71] OF BYTE;
		ST20_2_TZ535_PN_In_Out_32_byte_1 : ARRAY[0..31] OF BYTE;
		ST20_3_TZ535_PN_In_Out_32_byte_1 : ARRAY[0..31] OF BYTE;
		ST20_4_TZ535_PN_In_Out_32_byte_1 : ARRAY[0..31] OF BYTE;
		ST20_5_TZ535_PN_In_Out_32_byte_1 : ARRAY[0..31] OF BYTE;
		ST20_ET200SP_CM_4xIO_Link_1 : ARRAY[0..31] OF BYTE;
		ST20_ET200SP_CM_4xIO_Link_2 : ARRAY[0..31] OF BYTE;
		ST20_ET200SP_DI_16x24VDC_ST_1 : WORD;
		ST20_ET200SP_DI_16x24VDC_ST_2 : WORD;
		ST20_ET200SP_DI_16x24VDC_ST_3 : WORD;
		ST20_ET200SP_DI_16x24VDC_ST_4 : WORD;
		ST20_2_Schunk_IN_4_Double_Words_1 : ARRAY[0..15] OF BYTE;
		ST20_5_Schunk_IN_4_Double_Words_1 : ARRAY[0..15] OF BYTE;
		ST20_2_DM260_PCB1_Acquisition_Status_1 : ARRAY[0..2] OF BYTE;
		ST20_2_DM260_PCB1_Results_Status_1 : BYTE;
		ST20_2_DM260_PCB1_Soft_Event_Control_1 : BYTE;
		ST20_2_DM260_PCB1_Result_Data_64_bytes_1 : ARRAY[0..71] OF BYTE;
		ST20_2_DM260_PCB2_Acquisition_Status_1 : ARRAY[0..2] OF BYTE;
		ST20_2_DM260_PCB2_Results_Status_1 : BYTE;
		ST20_2_DM260_PCB2_Soft_Event_Control_1 : BYTE;
		ST20_2_DM260_PCB2_Result_Data_64_bytes_1 : ARRAY[0..71] OF BYTE;
		ST20_3_Schunk_IN_4_Double_Words_1 : ARRAY[0..15] OF BYTE;
		ST20_4_Schunk_IN_4_Double_Words_1 : ARRAY[0..15] OF BYTE;
		ST20_1_md_u2xxx_Machine_Status_1 : DWORD;
		ST20_1_md_u2xxx_Function_Status_1 : DWORD;
		ST20_1_md_u2xxx_Completion_Status_1 : ARRAY[0..7] OF BYTE;
		ST20_1_md_u2xxx_Error_Status_1 : ARRAY[0..7] OF BYTE;
		ST20_1_md_u2xxx_Error_Codes_1 : ARRAY[0..7] OF BYTE;
		ST20_1_md_u2xxx_Operate_Parametere_1 : ARRAY[0..15] OF BYTE;
		ST20_1_md_u2xxx_2D_Code_Read_Result_1 : ARRAY[0..7] OF BYTE;
		ST20_1_md_u2xxx_Count_Result_Data_1 : DWORD;
		ST20_1_md_u2xxx_Result_Data_128byte_1 : ARRAY[0..129] OF BYTE;
	END_STRUCT;
END_TYPE

(* ---- PlcOutputs.st ---- *)
TYPE
	PlcOutputs : STRUCT
		ST20_CPX_MPA1S_VMPA1_FB_EMS_8_8DO_1 : BYTE;
		ST20_CPX_MPA1S_VMPA1_FB_EMS_8_8DO_2 : BYTE;
		ST20_CPX_MPA1S_VMPA1_FB_EMS_8_8DO_3 : BYTE;
		ST20_CPX_MPA1S_VMPA1_FB_EMS_8_8DO_4 : BYTE;
		ST20_CPX_MPA1G_VMPA1_FB_EMG_8_8DO_1 : BYTE;
		ST20_6_Promess_Menu_30_33_Out_1 : WORD;
		ST20_6_Promess_Menu_30_34_Out_1 : WORD;
		ST20_6_Promess_Menu_30_35_Out_1 : WORD;
		ST20_6_Promess_Menu_30_36_Out_1 : WORD;
		ST20_6_Promess_Menu_30_37_Out_1 : WORD;
		ST20_6_Promess_Menu_30_38_Out_1 : WORD;
		ST20_6_Promess_Menu_30_39_Out_1 : WORD;
		ST20_6_Promess_Menu_30_40_Out_1 : WORD;
		ST20_6_Promess_Menu_30_41_Out_1 : WORD;
		ST20_6_Promess_Menu_30_42_Out_1 : WORD;
		ST20_6_Promess_Menu_30_43_Out_1 : WORD;
		ST20_6_Promess_Menu_30_44_Out_1 : WORD;
		ST20_6_Promess_Menu_30_45_Out_1 : WORD;
		ST20_6_Promess_Menu_30_46_Out_1 : WORD;
		ST20_6_Promess_Menu_30_47_Out_1 : WORD;
		ST20_6_Promess_Menu_30_48_Out_1 : WORD;
		ST20_6_Promess_Menu_30_49_Out_1 : WORD;
		ST20_6_Promess_Menu_30_50_Out_1 : WORD;
		ST20_6_Promess_Menu_30_51_Out_1 : WORD;
		ST20_6_Promess_Menu_30_52_Out_1 : WORD;
		ST20_6_Promess_Menu_30_53_Out_1 : WORD;
		ST20_6_Promess_Menu_30_54_Out_1 : WORD;
		ST20_6_Promess_Menu_30_55_Out_1 : WORD;
		ST20_6_Promess_Menu_30_56_Out_1 : WORD;
		ST20_6_Promess_Menu_30_57_Out_1 : WORD;
		ST20_6_Promess_Menu_30_58_Out_1 : WORD;
		ST20_6_Promess_Menu_30_59_Out_1 : WORD;
		ST20_6_Promess_Menu_30_60_Out_1 : WORD;
		ST20_6_Promess_Menu_30_61_Out_1 : WORD;
		ST20_6_Promess_Menu_30_62_Out_1 : WORD;
		ST20_6_Promess_Menu_30_63_Out_1 : WORD;
		ST20_6_Promess_Menu_30_64_Out_1 : WORD;
		ST20_7_CMMT_3GF1_DO_SERVO_1_Siemens_telegram_111_PZD_12_12 : ARRAY[0..23] OF BYTE;
		ST20_1_DM260_Acquisition_Control_1 : BYTE;
		ST20_1_DM260_Results_Control_1 : BYTE;
		ST20_1_DM260_Soft_Event_Control_1 : BYTE;
		ST20_1_DM260_User_Data_64_bytes_1 : ARRAY[0..67] OF BYTE;
		ST20_5_DM260_Acquisition_Control_1 : BYTE;
		ST20_5_DM260_Results_Control_1 : BYTE;
		ST20_5_DM260_Soft_Event_Control_1 : BYTE;
		ST20_5_DM260_User_Data_64_bytes_1 : ARRAY[0..67] OF BYTE;
		ST20_2_DM260_Acquisition_Control_1 : BYTE;
		ST20_2_DM260_Results_Control_1 : BYTE;
		ST20_2_DM260_Soft_Event_Control_1 : BYTE;
		ST20_2_DM260_User_Data_64_bytes_1 : ARRAY[0..67] OF BYTE;
		ST20_2_TZ535_PN_In_Out_32_byte_1 : ARRAY[0..31] OF BYTE;
		ST20_3_TZ535_PN_In_Out_32_byte_1 : ARRAY[0..31] OF BYTE;
		ST20_4_TZ535_PN_In_Out_32_byte_1 : ARRAY[0..31] OF BYTE;
		ST20_5_TZ535_PN_In_Out_32_byte_1 : ARRAY[0..31] OF BYTE;
		ST20_ET200SP_CM_4xIO_Link_1 : ARRAY[0..31] OF BYTE;
		ST20_ET200SP_CM_4xIO_Link_2 : ARRAY[0..31] OF BYTE;
		ST20_ET200SP_DQ_16x24VDC_0_5A_ST_1 : WORD;
		ST20_ET200SP_DQ_16x24VDC_0_5A_ST_2 : WORD;
		ST20_ET200SP_DQ_16x24VDC_0_5A_ST_3 : WORD;
		ST20_2_Schunk_OUT_4_Double_Words_1 : ARRAY[0..15] OF BYTE;
		ST20_5_Schunk_OUT_4_Double_Words_1 : ARRAY[0..15] OF BYTE;
		ST20_2_DM260_PCB1_Acquisition_Control_1 : BYTE;
		ST20_2_DM260_PCB1_Results_Control_1 : BYTE;
		ST20_2_DM260_PCB1_Soft_Event_Control_1 : BYTE;
		ST20_2_DM260_PCB1_User_Data_64_bytes_1 : ARRAY[0..67] OF BYTE;
		ST20_2_DM260_PCB2_Acquisition_Control_1 : BYTE;
		ST20_2_DM260_PCB2_Results_Control_1 : BYTE;
		ST20_2_DM260_PCB2_Soft_Event_Control_1 : BYTE;
		ST20_2_DM260_PCB2_User_Data_64_bytes_1 : ARRAY[0..67] OF BYTE;
		ST20_CPX_2_MPA1S_VMPA1_FB_EMS_8_8DO_1 : BYTE;
		ST20_CPX_2_MPA1S_VMPA1_FB_EMS_8_8DO_2 : BYTE;
		ST20_CPX_2_MPA1G_VMPA1_FB_EMG_8_8DO_1 : BYTE;
		ST20_CPX_2_MPA1G_VMPA1_FB_EMG_8_8DO_2 : BYTE;
		ST20_3_Schunk_OUT_4_Double_Words_1 : ARRAY[0..15] OF BYTE;
		ST20_4_Schunk_OUT_4_Double_Words_1 : ARRAY[0..15] OF BYTE;
		ST20_1_md_u2xxx_General_Request_1 : ARRAY[0..7] OF BYTE;
		ST20_1_md_u2xxx_Function_Request_1 : DWORD;
		ST20_1_md_u2xxx_Request_Completion_Clear_1 : ARRAY[0..7] OF BYTE;
		ST20_1_md_u2xxx_Request_Parameter_1 : DWORD;
		ST20_1_md_u2xxx_Request_Data_128byte_1 : ARRAY[0..129] OF BYTE;
	END_STRUCT;
END_TYPE
